// TIA Portal V20 program export: 1 tag tables, 0 data types, 0 data blocks, 2 code blocks (in call order from the OBs), 0 instance data blocks

VAR_GLOBAL   // PLC tag table "Default tag table"
   Start AT %I0.0 : Bool;
   Stop AT %I0.1 : Bool;
   Process_on AT %Q0.0 : Bool;
   AutoON AT %M100.0 : Bool;   // AutoON
END_VAR

ORGANIZATION_BLOCK "Main"   // OB1, LAD, ProgramCycle
TITLE = "Main Program Sweep (Cycle)"
{ S7_Optimized_Access := 'TRUE' }
// stored: SetENOAutomatically false
   VAR_INPUT
      Initial_Call : Bool;   // Initial call of this OB
      Remanence : Bool;   // =True, if remanent data are available
   END_VAR
   VAR_TEMP   // added for the SCL form of the ladder/FBD networks
      _w1 : Bool;
   END_VAR
BEGIN

REGION Network 1
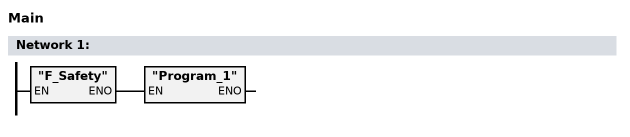
   RUNG wire#powerrail
      "F_Safety"()
      "Program_1"()
   END_RUNG
   // the same network as SCL:
   "F_Safety"(ENO => #_w1);
   IF #_w1 THEN "Program_1"(); END_IF;
END_REGION
END_ORGANIZATION_BLOCK

FUNCTION "Program_1" : Void   // FC1, LAD
{ S7_Optimized_Access := 'TRUE' }
// stored: SetENOAutomatically false
BEGIN

REGION Network 1
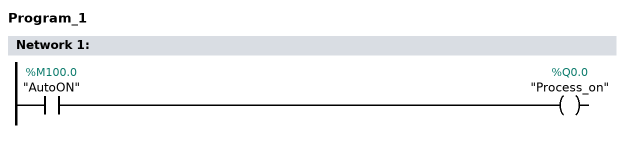
   RUNG wire#powerrail
      Contact( "AutoON" )
      Coil( "Process_on" )
   END_RUNG
   // the same network as SCL:
   "Process_on" := "AutoON";
END_REGION
END_FUNCTION
